// TwinCAT 3 PLC project PLC1
// Title: AutomationBaseClasses
// Company: PTW TU Darmstadt
// Author: Fabian Borst, Lukas Theisinger, Michael Frank, Tobias Lademann
// ProjectVersion: 1.1
// ProgramVersion: 3.1.4023.0
// libraries:
//   Tc2_ControllerToolbox, * (Beckhoff Automation GmbH)
//   Tc2_MBus, * (Beckhoff Automation GmbH)
//   Tc2_ModbusSrv, * (Beckhoff Automation GmbH)
//   Tc2_Standard, * (Beckhoff Automation GmbH)
//   Tc2_System, * (Beckhoff Automation GmbH)
//   Tc2_Utilities, * (Beckhoff Automation GmbH)
//   Tc3_Module, * (Beckhoff Automation GmbH)
// project tree:
//   DUTs/0 Base Data Structs/ E_SystemControlState.TcDUT, E_SystemOperatingState.TcDUT, ST_Control.TcDUT (not stored), ST_ControlState.TcDUT, ST_SensorState.TcDUT, ST_SetPointState.TcDUT, ST_SetSetPoint.TcDUT, ST_SystemState.TcDUT
//   DUTs/1 Actor Data Structs/DicreteValve/ E_DiscreteValveFeedbackMode.TcDUT, E_DiscreteValvePosition.TcDUT, ST_DiscreteValveDefaultParameters.TcDUT, ST_DiscreteValveState.TcDUT
//   DUTs/1 Actor Data Structs/MixingValve/ E_MixingValveControlMode.TcDUT, ST_MixingValveDefaultParameters.TcDUT, ST_MixingValveSetParameters.TcDUT
//   DUTs/1 Actor Data Structs/Pumps/ E_GrundfosMagna3ControlMode.TcDUT, ST_PumpGrundfosMagna3DefaultParameters.TcDUT, ST_PumpGrundfosMagna3Genibus.TcDUT, ST_PumpGrundfosMagna3SetParameters.TcDUT, ST_PumpGrundfosMagna3State.TcDUT
//   DUTs/2 Sensor Data Structs/ ST_ElectricityMeterState.TcDUT, ST_EmonioP3DefaultParameters.TcDUT, ST_EmonioP3State.TcDUT, ST_GasMeterDefaultParameters.TcDUT, ST_MollineC3HeatCounterState.TcDUT, ST_GasMeterState.TcDUT, ST_MollineC3HeatCounterDefaultParameters.TcDUT, ST_StarkMultical302HeatCounterState.TcDUT, ST_TemperatureSensorDefaultParameters.TcDUT (not stored)
//   DUTs/3 Utility Data Structs/ ST_RangeCheckDefaultParameters.TcDUT, ST_ClockDefaultParameters.TcDUT (not stored), ST_ClockState.TcDUT (not stored)
//   POUs/2 Sensors/ FB_ElectricityMeter_ABBA44113100.TcPOU, FB_ElectricityMeter_BergDCMI461WP.TcPOU, FB_ElectricityMeter_ABBA44213100.TcPOU, FB_EmonioP3.TcPOU, FB_GasMeter_Aerius_G4.TcPOU, FB_MollineEHeatCounter.TcPOU, FB_MollineUltramess403HeatCounter.TcPOU, FB_PressureSensor.TcPOU, FB_StarkMultical302HeatCounter.TcPOU, FB_TemperatureSensor_KL3214.TcPOU, FB_MollineC3HeatCounter.TcPOU, FB_TemperatureSensor.TcPOU
//   POUs/3 Utilities/0 Base/ FB_RangeCheck.TcPOU, FB_Clock.TcPOU, Limiter.TcPOU
//   POUs/3 Utilities/2 Profibus/ ConvertBitToByte.TcPOU, ConvertByteToBit.TcPOU (not stored), FB_Genibus.TcPOU, BufferIntToReal.TcPOU (not stored), BufferRealToReal.TcPOU (not stored), BufferUdintToReal.TcPOU
//   POUs/0 Base Classes/ FB_Actuator2Point.TcPOU, FB_ActuatorContinous.TcPOU, FB_Sensor.TcPOU, FB_SystemContinous.TcPOU
//   POUs/1 Actors/ FB_DiscreteValve.TcPOU, FB_PumpGrundfosMagna3.TcPOU, FB_MixingValve.TcPOU
//   POUs/3 Utilities/1 AI_AO/ FB_AnalogInput.TcPOU (not stored), FB_AnalogOutput.TcPOU
// real-time tasks:
//   TASK TaskMAIN: cycle T#10ms, priority 20, ADS port 350

// ---- DUTs/0 Base Data Structs/E_SystemControlState.TcDUT
{attribute 'qualified_only'}
{attribute 'strict'}
TYPE E_SystemControlState :
(
	automatic 	:= 0,
	algorithm	:= 1,
	manual		:= 2
);
END_TYPE

// ---- DUTs/0 Base Data Structs/E_SystemOperatingState.TcDUT
{attribute 'qualified_only'}
{attribute 'strict'}
TYPE E_SystemOperatingState :
(
	standby 	:= 0,
	rampUp		:= 1,
	rampDown	:= 2,
	operational	:= 3,
	working		:= 4
);
END_TYPE

// ---- DUTs/0 Base Data Structs/ST_ControlState.TcDUT
{attribute 'OPC.UA.DA.StructuredType' := '1'}
TYPE ST_ControlState :
STRUCT
	bStatusOn 		: BOOL; //status on / off
	sAccessMode		: STRING; //current access mode as string
	nAccessmode		: E_SystemControlState; //current access mode (1 = automatic, 2 = algorihm, 3 = manual)
END_STRUCT
END_TYPE

// ---- DUTs/0 Base Data Structs/ST_SensorState.TcDUT
{attribute 'OPC.UA.DA.StructuredType' := '1'}
TYPE ST_SensorState :
STRUCT
	fValue 		: REAL; //current value
	sUnit		: STRING; //current unit of sensor value
END_STRUCT
END_TYPE

// ---- DUTs/0 Base Data Structs/ST_SetPointState.TcDUT
{attribute 'OPC.UA.DA.StructuredType' := '1'}
TYPE ST_SetPointState :
STRUCT
	fOperatingPoint		: REAL; //current operating point
	fSetPoint			: REAL; //current set point
	sSetPointUnit		: STRING; //current set point unit
	sOperatingPointUnit : STRING; //current operating point unit 
	aSetPointLimits		: ARRAY[1..2] OF REAL; //lower and upper limit of setpoint
END_STRUCT
END_TYPE

// ---- DUTs/0 Base Data Structs/ST_SetSetPoint.TcDUT
{attribute 'OPC.UA.DA.StructuredType' := '1'}
TYPE ST_SetSetPoint :
STRUCT
	fSetPointAlgorithm		 : REAL; //set setpoint in percent 0.0 - 100.0
	fSetPointManual			 : REAL; //set setpoint in percent 0.0 - 100.0
END_STRUCT
END_TYPE

// ---- DUTs/0 Base Data Structs/ST_SystemState.TcDUT
{attribute 'OPC.UA.DA.StructuredType' := '1'}
TYPE ST_SystemState :
STRUCT
	sOperatingState : STRING; //operating state as string
	nOperatingState : E_SystemOperatingState; //operating state as integer
	bError : BOOL; //true if there is an error in any system component
END_STRUCT
END_TYPE

// ---- DUTs/1 Actor Data Structs/DicreteValve/E_DiscreteValveFeedbackMode.TcDUT
{attribute 'qualified_only'}
{attribute 'strict'}
TYPE E_DiscreteValveFeedbackMode :
(
	noFeedback := 0, //no feedback signal about valve position available
	openedFeedback := 1, //feedback signal if valve is open
	closedFeedback := 2, //feedback signal if valve is closed
	dualFeedback := 3 //feedback signal if valve is open/closed
);
END_TYPE

// ---- DUTs/1 Actor Data Structs/DicreteValve/E_DiscreteValvePosition.TcDUT
{attribute 'qualified_only'}
{attribute 'strict'}
TYPE E_DiscreteValvePosition :
(	
	noValidInformation := 0, //no information about position available
	moving := 1, //valve is moving
	closed := 2, //valve is closed
	open := 3 //valve is open
);
END_TYPE

// ---- DUTs/1 Actor Data Structs/DicreteValve/ST_DiscreteValveDefaultParameters.TcDUT
TYPE ST_DiscreteValveDefaultParameters :
STRUCT
	nFeedback : E_DiscreteValveFeedbackMode; //valve feedback mode as integer
END_STRUCT
END_TYPE

// ---- DUTs/1 Actor Data Structs/DicreteValve/ST_DiscreteValveState.TcDUT
TYPE ST_DiscreteValveState :
STRUCT
	nPosition : E_DiscreteValvePosition; //valve feedback mode as integer
END_STRUCT
END_TYPE

// ---- DUTs/1 Actor Data Structs/MixingValve/E_MixingValveControlMode.TcDUT
{attribute 'qualified_only'}
{attribute 'strict'}
TYPE E_MixingValveControlMode :
(
	position := 0, //control position
	heating := 1, //control temperature for heating application
	cooling := 2, //control temperature for cooling application
	thermalPower := 3 //control thermal power
);
END_TYPE

// ---- DUTs/1 Actor Data Structs/MixingValve/ST_MixingValveDefaultParameters.TcDUT
TYPE ST_MixingValveDefaultParameters:
STRUCT
	bFeedbackSignal : BOOL := TRUE; //true if valve gets a feedback signal for acual position
	fDefaultPosition : REAL := 0; //default position when bSetStatusOn = false
	fOffsetTerminal : REAL := 0; //voltage offset of terminal for input signal
	fControllerAmplification : LREAL := 0.265;
	tControllerIntegralTime : TIME := T#15S;
	fOutMaxLimit : LREAL := 100; //maximum output of controller
	fOutMinLimit : LREAL := 0; //minimum output of controller
	bARWOnIPartOnly : BOOL := TRUE; //if true, integration of I component stops, when integrator output reaches limit
	tTaskCycleTime	: TIME;
	tCtrlCycleTime	: TIME;
	aSetPointLimitsPosition	: ARRAY[1..2] OF REAL := [0,100]; //setpoint limits for position mode
	aSetPointLimitsTemperature : ARRAY[1..2] OF REAL := [0,100]; //setpoint limits for temperature mode
	aSetPointLimitsThermalPower : ARRAY[1..2] OF REAL := [-100,100]; //setpoint limits for heating and cooling power in kW
END_STRUCT
END_TYPE

// ---- DUTs/1 Actor Data Structs/MixingValve/ST_MixingValveSetParameters.TcDUT
{attribute 'OPC.UA.DA.StructuredType' := '1'}
TYPE ST_MixingValveSetParameters :
STRUCT
	nControlModeAlgorithm : E_MixingValveControlMode; //control mode in algorithm mode
	nControlModeManual : E_MixingValveControlMode; //control in manuel mode
END_STRUCT
END_TYPE

// ---- DUTs/1 Actor Data Structs/Pumps/E_GrundfosMagna3ControlMode.TcDUT
{attribute 'qualified_only'}
{attribute 'strict'}
TYPE E_GrundfosMagna3ControlMode :
(
	constantSpeed := 0, //constant speed control - 0.0 - 100.0 %
	constantTemperature_Heating := 1, //temperature control if flow is heated
	constantTemperature_Cooling := 2, //temperature control if flow is cooled
	temperatureDifference := 3, //temperature difference control
	pressureDifference := 4, //pressure difference control
	proportionalPressureControl := 5, //proportional pressure control
	thermalPower := 6 //thermal power control
);
END_TYPE

// ---- DUTs/1 Actor Data Structs/Pumps/ST_PumpGrundfosMagna3DefaultParameters.TcDUT
TYPE ST_PumpGrundfosMagna3DefaultParameters :
STRUCT
	bExternalTemperatureSensor 	: BOOL := TRUE; //pump measures beside the internal temperature als and external temperature
	bPumpBeforeApplication : BOOL := TRUE; //pump position before application
	fControllerAmplification : LREAL := 0.265;
	tControllerIntegralTime : TIME := T#15S;
	tTaskCycleTime	: TIME;
	tCtrlCycleTime	: TIME;	
	aSetPointLimits_constantSpeed : ARRAY[1..2] OF REAL := [0,100]; //degreeC
	aSetPointLimits_Temperature	: ARRAY[1..2] OF REAL := [0,100]; //degreeC
	aSetPointLimits_Pressure : ARRAY[1..2] OF REAL := [0,3]; //bar
	aSetPointLimitsThermalPower : ARRAY[1..2] OF REAL := [-100,100]; //setpoint limits for heating and cooling power in kW
	fMaximumVolumeFlowRate : REAL := 1.925; //default parameters for Magna3 25-40
	fNominalVolumeFlowRate : REAL := 0.000635; //default parameters for Magna3 25-40
	fMaximumPressureDifference : REAL := 40000; //default parameters for Magna3 25-40
END_STRUCT
END_TYPE

// ---- DUTs/1 Actor Data Structs/Pumps/ST_PumpGrundfosMagna3Genibus.TcDUT
TYPE ST_PumpGrundfosMagna3Genibus :
STRUCT
	SequenceNumber 	: BYTE;			(*SequenceNumber: Is the trigger, every time the value changes a new reply will be generated. *)
									(*For return telegram: values valid if Number matches request SquenceNumber*)
	DestAddress		: BYTE;			(*Address of GeniPro Slave, Broadcast = 16#FF*)
	Class			: BYTE;			(* no further Info provided*)
	OpLength		: BYTE; 		(* Operation and Length / for Reply Acknowledge and Length*)
	Data1			: BYTE;
	Data2			: BYTE;
	Data3			: BYTE;
	Data4			: BYTE;
	Data5			: BYTE;
END_STRUCT
END_TYPE

// ---- DUTs/1 Actor Data Structs/Pumps/ST_PumpGrundfosMagna3SetParameters.TcDUT
{attribute 'OPC.UA.DA.StructuredType' := '1'}
TYPE ST_PumpGrundfosMagna3SetParameters :
STRUCT
	nControlModeAlgorithm : E_GrundfosMagna3ControlMode; //control mode in algorithm mode
	nControlModeManual : E_GrundfosMagna3ControlMode; //control mode in manual mode
	bReset : BOOL; //resets errors and warnings
END_STRUCT
END_TYPE

// ---- DUTs/1 Actor Data Structs/Pumps/ST_PumpGrundfosMagna3State.TcDUT
{attribute 'OPC.UA.DA.StructuredType' := '1'}
TYPE ST_PumpGrundfosMagna3State :
STRUCT
	bRemoteControlOn : BOOL; //0 = control by pump, 1 = control by bus 	
	bError : BOOL; //true if pump shows an error
	bWarning : BOOL; //true if pump shows a warning
	sErrorMessage : STRING; //error code
	sWarningMessage : STRING; //warning code
	fVolumeFlowRate : REAL;
	sVolumeFlowRateUnit : STRING := 'm3/h';
	fTemperatureInternal : REAL; 
	sTemperatureInternalUnit : STRING := 'degreeC';
	fTemperatureExternal : REAL;
	sTemperatureExternalUnit : STRING := 'degreeC';
	fTemperatureDifference : REAL;
	sTemperatureDifferenceUnit: STRING := 'K';
	fPressureDifference : REAL;
	sPressureDifferenceUnit : STRING := 'Pa';
	fPowerElectric : REAL;
	sPowerElectricUnit : STRING := 'kW';
	fPowerHydraulic : REAL;
	sPowerHydraulicUnit : STRING := 'W';
	fPowerThermal : REAL;
	sPowerThermalUnit : STRING := 'W';
	fRotationalSpeed : REAL;
	sRotationalSpeedUnit : STRING := 'rpm';
END_STRUCT
END_TYPE

// ---- DUTs/2 Sensor Data Structs/ST_ElectricityMeterState.TcDUT
{attribute 'OPC.UA.DA.StructuredType' := '1'}
TYPE ST_ElectricityMeterState :
STRUCT
	fPower			: REAL;
	sPowerUnit		: STRING := 'kW';
	fWork			: REAL;
	sWorkUnit		: STRING := 'kWh';
END_STRUCT
END_TYPE

// ---- DUTs/2 Sensor Data Structs/ST_EmonioP3DefaultParameters.TcDUT
TYPE ST_EmonioP3DefaultParameters :
STRUCT
	fCalorificValue : REAL := 11.49;
END_STRUCT
END_TYPE

// ---- DUTs/2 Sensor Data Structs/ST_EmonioP3State.TcDUT
{attribute 'OPC.UA.DA.StructuredType' := '1'}
TYPE ST_EmonioP3State :
STRUCT
	fPower 					: REAL;
	sPowerUnit				: STRING := 'kW';
	fVoltage 				: REAL;
	sVoltageUnit			: STRING := 'V';
	fCurrent				: REAL;
	sCurrentUnit			: STRING := 'A';
	fEnergy					: REAL;
	sEnergyUnit				: STRING := 'kWh';
	fTemperature			: REAL;
	sTemperatureUnit		: STRING := 'degreeC';
	fPulse					: REAL;
	sPulse					: STRING := 'm^3';
	fPulseGasPower			: REAL;
	sPulseGasPower			: STRING := 'kW';
END_STRUCT
END_TYPE

// ---- DUTs/2 Sensor Data Structs/ST_GasMeterDefaultParameters.TcDUT
TYPE ST_GasMeterDefaultParameters :
STRUCT
	fCalorificValue : REAL := 11.49;
END_STRUCT
END_TYPE

// ---- DUTs/2 Sensor Data Structs/ST_MollineC3HeatCounterState.TcDUT
{attribute 'OPC.UA.DA.StructuredType' := '1'}
TYPE ST_MollineC3HeatCounterState :
STRUCT
	fVolume						: REAL;
	sVolumeUnit					: STRING := 'm3';
	fFeedTemperature			: REAL;
	sFeedTemperatureUnit		: STRING := 'degreeC';
	fReturnTemperature			: REAL;
	sReturnTemperatureUnit		: STRING := 'degreeC';
	fVolumeFlowRate				: REAL;
	sVolumeFlowRateUnit			: STRING := 'm3/h';
	fHeatEnergy					: REAL;
	sHeatEnergyUnit				: STRING := 'MWh';
	fHeatFlowRate				: REAL;
	sHeatFlowRateUnit			: STRING := 'kW';
	fTemperatureDifference		: REAL;
	sTemperatureDifferenceUnit 	: STRING := 'K';
END_STRUCT
END_TYPE

// ---- DUTs/2 Sensor Data Structs/ST_GasMeterState.TcDUT
{attribute 'OPC.UA.DA.StructuredType' := '1'}
TYPE ST_GasMeterState :
STRUCT
	fVolume					: REAL;
	sVolumeUnit				: STRING := 'm3';
	fTemperature			: REAL;
	sTemperatureUnit		: STRING := 'degreeC';
	fVolumeFlowRate			: REAL;
	sVolumeFlowRateUnit		: STRING := 'm3/h';
	fPower 					: REAL;
	sPowerUnit				: STRING := 'kW';
END_STRUCT
END_TYPE

// ---- DUTs/2 Sensor Data Structs/ST_MollineC3HeatCounterDefaultParameters.TcDUT
TYPE ST_MollineC3HeatCounterDefaultParameters:
STRUCT
	fSpecificHeatCapacity : REAL := 4.19;
END_STRUCT
END_TYPE

// ---- DUTs/2 Sensor Data Structs/ST_StarkMultical302HeatCounterState.TcDUT
{attribute 'OPC.UA.DA.StructuredType' := '1'}
TYPE ST_StarkMultical302HeatCounterState :
STRUCT
	fVolume						: REAL;
	sVolumeUnit					: STRING := 'm3';
	fFeedTemperature			: REAL;
	sFeedTemperatureUnit		: STRING := 'degreeC';
	fReturnTemperature			: REAL;
	sReturnTemperatureUnit		: STRING := 'degreeC';
	fVolumeFlowRate				: REAL;
	sVolumeFlowRateUnit			: STRING := 'm3/h';
	fHeatEnergy					: REAL;
	sHeatEnergyUnit				: STRING := 'MWh';
	fHeatFlowRate				: REAL;
	sHeatFlowRateUnit			: STRING := 'kW';
	fTemperatureDifference		: REAL;
	sTemperatureDifferenceUnit 	: STRING := 'K';
END_STRUCT
END_TYPE

// ---- DUTs/3 Utility Data Structs/ST_RangeCheckDefaultParameters.TcDUT
TYPE ST_RangeCheckDefaultParameters :
STRUCT
	fRestoreDifference : REAL; //difference to upper or lower limit to restore algorithm permission
	tTaskCycleTime : TIME;
	tCtrlCycleTime : TIME;
END_STRUCT
END_TYPE

// ---- POUs/2 Sensors/FB_ElectricityMeter_ABBA44113100.TcPOU
FUNCTION_BLOCK FB_ElectricityMeter_ABBA44113100
VAR_INPUT
	aElectricityMeterTelegramm	: ARRAY[1..cMBUS_MaxTelegrams] OF ST_MBus_Data2;
END_VAR
VAR_OUTPUT
	fWork : REAL; //Wh
	fPower : REAL; //W
END_VAR
VAR
	{attribute 'OPC.UA.DA' := '1'}
	sensorState : ST_ElectricityMeterState;
END_VAR

sensorState.fWork := STRING_TO_REAL(aElectricityMeterTelegramm[1].arrData[1].sValue)/1000;
sensorState.fPower := STRING_TO_REAL(aElectricityMeterTelegramm[2].arrData[1].sValue)/1000;

fWork := sensorState.fWork;
fPower := sensorState.fPower;

END_FUNCTION_BLOCK

// ---- POUs/2 Sensors/FB_ElectricityMeter_BergDCMI461WP.TcPOU
FUNCTION_BLOCK FB_ElectricityMeter_BergDCMI461WP
VAR_INPUT
	aElectricityMeterTelegramm	: ARRAY[1..cMBUS_MaxTelegrams] OF ST_MBus_Data2;
END_VAR
VAR_OUTPUT
	fWork : REAL; //Wh
	fPower : REAL; //W
END_VAR
VAR
	{attribute 'OPC.UA.DA' := '1'}
	sensorState : ST_ElectricityMeterState;
END_VAR

sensorState.fWork := STRING_TO_REAL(aElectricityMeterTelegramm[1].arrData[1].sValue)/1000;
sensorState.fPower := STRING_TO_REAL(aElectricityMeterTelegramm[1].arrData[2].sValue)/1000;

//set outputs
fWork := sensorState.fWork;
fPower := sensorState.fPower;

END_FUNCTION_BLOCK

// ---- POUs/2 Sensors/FB_ElectricityMeter_ABBA44213100.TcPOU
FUNCTION_BLOCK FB_ElectricityMeter_ABBA44213100
VAR_INPUT
	aElectricityMeterTelegramm	: ARRAY[1..cMBUS_MaxTelegrams] OF ST_MBus_Data2;
END_VAR
VAR_OUTPUT
	fWork : REAL; //Wh
	fPower : REAL; //W
END_VAR
VAR
	{attribute 'OPC.UA.DA' := '1'}
	sensorState : ST_ElectricityMeterState;
END_VAR

sensorState.fWork := STRING_TO_REAL(aElectricityMeterTelegramm[1].arrData[1].sValue)/1000;
sensorState.fPower := STRING_TO_REAL(aElectricityMeterTelegramm[2].arrData[2].sValue)/1000;

//set outputs
fWork := sensorState.fWork;
fPower := sensorState.fPower;

END_FUNCTION_BLOCK

// ---- POUs/2 Sensors/FB_EmonioP3.TcPOU
FUNCTION_BLOCK FB_EmonioP3
VAR_INPUT
	sIPAddr : STRING(15);
END_VAR
VAR_OUTPUT
	fPower : REAL; 			//kW
	fVoltage : REAL; 		//V
	fCurrent : REAL; 		//A
	fEnergy : REAL; 		//kWh
	fTemperature : REAL; 	//°C
	fPulse : REAL; 			//m^3
	fPulseGasPower : REAL;	//kW
	
	bErrorEM: BOOL;
	bErrorTemp: BOOL;
	bErrorPulse : BOOL;
END_VAR
VAR
	{attribute 'OPC.UA.DA' := '1'}
	sensorState : ST_EmonioP3State;
	
	localDefaultParameters : ST_EmonioP3DefaultParameters;
	
	fbEmonioElectricity : FB_MBReadRegs;
	fbEmonioTemperature : FB_MBReadRegs;
	fbEmonioPulse : FB_MBReadRegs;
	
	//timer to execute modbus fb
	Timer : TON;	
	bStartTimer : BOOL;
	bReadModbus : BOOL;
	
	arrInputRegsElectricity: ARRAY[0..13] OF WORD;			  // buffer for modbus fb electricity values
	arrInputRegsTemperature: ARRAY[0..1] OF WORD;			  // buffer for modbus fb temperature value
	arrInputRegsPulse: ARRAY[0..1] OF WORD;			  // buffer for modbus fb pulse value
	
    nErrIdEM: UDINT;
    nErrIdTemp: UDINT;
	nErrIdPulse: UDINT;
	
	//define arrays to convert from 16-bit word to real values
	PowerArray: ARRAY [0..1] OF WORD;
	VoltageArray: ARRAY [0..1] OF WORD;
	CurrentArray: ARRAY [0..1] OF WORD;
	EnergyArray: ARRAY [0..1] OF WORD;
	TemperatureArray: ARRAY [0..1] OF WORD;
	PulseArray: ARRAY [0..1] OF WORD;
	
	PowerInWatt : REAL; //helper variable to convert from W to kW
	
	//timer to execute modbus fb
	TimerGas : TON;	
	bStartTimerGas : BOOL;
	fPulseLastValue : REAL;
END_VAR

//Start and check timer for 2s interval
Timer(IN := bStartTimer,
	PT := T#2S);
bStartTimer := TRUE;
IF Timer.Q THEN
	bReadModbus := TRUE;
	bStartTimer := FALSE;	
END_IF

// Read Emonio via Modbus
fbEmonioElectricity(    
	sIPAddr := sIPAddr,   			//IP adress of the device
	nTCPPort := 502,				//Port number of the target device
	nUnitID := 255,					//Identification number of a serial sub-network device
	nQuantity  := 13,				//Number of input registers (data words) to be read
	nMBAddr := 300,					// Start address of the output registers to be read (word offset)
	cbLength := SIZEOF(arrInputRegsElectricity),
	pDestAddr := ADR(arrInputRegsElectricity),
	bExecute := bReadModbus,         // trigger
	tTimeout  := T#20S,
	bError => bErrorEM,				// Error handling
	nErrId => nErrIdEM				// Error handling 
);

fbEmonioTemperature(    
	sIPAddr := sIPAddr,   			//IP adress of the device
	nTCPPort := 502,				//Port number of the target device
	nUnitID := 255,					//Identification number of a serial sub-network device
	nQuantity  := 2,				//Number of input registers (data words) to be read
	nMBAddr := 500,					// Start address of the output registers to be read (word offset)
	cbLength := SIZEOF(arrInputRegsTemperature),
	pDestAddr := ADR(arrInputRegsTemperature),
	bExecute := bReadModbus,         // trigger
	tTimeout  := T#20S,
	bError => bErrorTemp,				// Error handling
	nErrId => nErrIdTemp				// Error handling 
);

fbEmonioPulse(    
	sIPAddr := sIPAddr,   			//IP adress of the device
	nTCPPort := 502,				//Port number of the target device
	nUnitID := 255,					//Identification number of a serial sub-network device
	nQuantity  := 2,				//Number of input registers (data words) to be read
	nMBAddr := 800,					// Start address of the output registers to be read (word offset)
	cbLength := SIZEOF(arrInputRegsPulse),
	pDestAddr := ADR(arrInputRegsPulse),
	bExecute := bReadModbus,         // trigger
	tTimeout  := T#20S,
	bError => bErrorPulse,				// Error handling
	nErrId => nErrIdPulse				// Error handling 
);

bReadModbus := FALSE;

//create arrays with word outputs
PowerArray[0] := arrInputRegsElectricity[4];
PowerArray[1] := arrInputRegsElectricity[5];
VoltageArray[0] := arrInputRegsElectricity[0];
VoltageArray[1] := arrInputRegsElectricity[1];
CurrentArray[0] := arrInputRegsElectricity[2];
CurrentArray[1] := arrInputRegsElectricity[3];
EnergyArray[0] := arrInputRegsElectricity[12];
EnergyArray[1] := arrInputRegsElectricity[13];
TemperatureArray[0] := arrInputRegsTemperature[0];
TemperatureArray[1] := arrInputRegsTemperature[1];
PulseArray[0] := arrInputRegsPulse[0];
PulseArray[1] := arrInputRegsPulse[1];

//convert word to real values
MEMCPY(ADR(PowerInWatt), ADR(PowerArray), 4);
sensorState.fPower := PowerInWatt/1000;
MEMCPY(ADR(sensorState.fVoltage), ADR(VoltageArray), 4);
MEMCPY(ADR(sensorState.fCurrent), ADR(CurrentArray), 4);
MEMCPY(ADR(sensorState.fEnergy), ADR(EnergyArray), 4);
MEMCPY(ADR(sensorState.fTemperature), ADR(TemperatureArray), 4);
MEMCPY(ADR(sensorState.fPulse), ADR(PulseArray), 4);

TimerGas(IN := bStartTimerGas,
	PT := T#30S);
bStartTimerGas := TRUE;

//overwrite last value durint init as long as last value remains zero
IF fPulseLastValue = 0 THEN
	fPulseLastValue := fPulse;
END_IF
IF TimerGas.Q THEN
	sensorState.fPulseGasPower := (fPulse-fPulseLastValue)*120*localDefaultParameters.fCalorificValue; //Gas power in kW
	fPulseLastValue := fPulse;
	bStartTimerGas := FALSE;	
END_IF

//define output variables
fPower := sensorState.fPower;
fVoltage := sensorState.fVoltage;
fCurrent := sensorState.fCurrent;
fEnergy := sensorState.fEnergy;
fTemperature := sensorState.fTemperature;
fPulse := sensorState.fPulse;
fPulseGasPower := sensorState.fPulseGasPower;

END_FUNCTION_BLOCK

// ---- POUs/2 Sensors/FB_GasMeter_Aerius_G4.TcPOU
FUNCTION_BLOCK FB_GasMeter_Aerius_G4
VAR_INPUT
	aGasmeterTelegramm	: ARRAY[1..cMBUS_MaxTelegrams] OF ST_MBus_Data2;
END_VAR
VAR_OUTPUT
	fVolumeFlowRate : REAL; //m3/h
	fTemperature : REAL; //°C
END_VAR
VAR
	{attribute 'OPC.UA.DA' := '1'}
	sensorState : ST_GasMeterState;
	
	localDefaultParameters : ST_GasMeterDefaultParameters;
END_VAR

sensorState.fTemperature := STRING_TO_REAL(aGasmeterTelegramm[1].arrData[3].sValue);
sensorState.fVolumeFlowRate := STRING_TO_REAL(aGasmeterTelegramm[1].arrData[2].sValue);
sensorState.fVolume := STRING_TO_REAL(aGasmeterTelegramm[1].arrData[1].sValue);
sensorState.fPower := sensorState.fVolumeFlowRate*localDefaultParameters.fCalorificValue; //calculate Power in kW

//set outputs
fVolumeFlowRate := sensorState.fVolume;
fTemperature := sensorState.fTemperature;

END_FUNCTION_BLOCK

// ---- POUs/2 Sensors/FB_MollineEHeatCounter.TcPOU
FUNCTION_BLOCK FB_MollineEHeatCounter
VAR_INPUT
	aHeatCounterTelegramm : ARRAY[1..cMBUS_MaxTelegrams] OF ST_MBus_Data2;
END_VAR
VAR_OUTPUT
	fFeedTemperature : REAL; //°C
	fReturnTemperature : REAL; //°C
	fVolumeFlowRate : REAL; //m3/h
	fHeatFlowRate : REAL; //kW
END_VAR
VAR
	{attribute 'OPC.UA.DA' := '1'}
	sensorState : ST_MollineC3HeatCounterState;
END_VAR

//set sensor state
sensorState.fVolume := STRING_TO_REAL(aHeatCounterTelegramm[1].arrData[3].sValue);
sensorState.fFeedTemperature := STRING_TO_REAL(aHeatCounterTelegramm[1].arrData[7].sValue);
sensorState.fReturnTemperature := STRING_TO_REAL(aHeatCounterTelegramm[1].arrData[8].sValue);
sensorState.fVolumeFlowRate := STRING_TO_REAL(aHeatCounterTelegramm[1].arrData[6].sValue);
sensorState.fHeatEnergy := STRING_TO_REAL(aHeatCounterTelegramm[1].arrData[2].sValue)/1000000;
sensorState.fTemperatureDifference := STRING_TO_REAL(aHeatCounterTelegramm[1].arrData[9].sValue);

//calculate fHeatFlowRate because heat meter does not measure negative flows
sensorState.fHeatFlowRate := sensorState.fVolumeFlowRate/3.6*4.19*sensorState.fTemperatureDifference;

//set outputs
fFeedTemperature := sensorState.fFeedTemperature;
fReturnTemperature := sensorState.fReturnTemperature;
fVolumeFlowRate := sensorState.fVolumeFlowRate;
fHeatFlowRate := sensorState.fHeatFlowRate;

END_FUNCTION_BLOCK

// ---- POUs/2 Sensors/FB_MollineUltramess403HeatCounter.TcPOU
FUNCTION_BLOCK FB_MollineUltramess403HeatCounter
VAR_INPUT
	aHeatCounterTelegramm : ARRAY[1..cMBUS_MaxTelegrams] OF ST_MBus_Data2;
END_VAR
VAR_OUTPUT
	fFeedTemperature : REAL; //°C
	fReturnTemperature : REAL; //°C
	fVolumeFlowRate : REAL; //m3/h
	fHeatFlowRate : REAL; //kW
END_VAR
VAR
	{attribute 'OPC.UA.DA' := '1'}
	sensorState : ST_MollineC3HeatCounterState;
END_VAR

//set sensor state
sensorState.fVolume := STRING_TO_REAL(aHeatCounterTelegramm[1].arrData[5].sValue);
sensorState.fFeedTemperature := STRING_TO_REAL(aHeatCounterTelegramm[1].arrData[11].sValue);
sensorState.fReturnTemperature := STRING_TO_REAL(aHeatCounterTelegramm[1].arrData[12].sValue);
sensorState.fVolumeFlowRate := STRING_TO_REAL(aHeatCounterTelegramm[1].arrData[17].sValue);
sensorState.fHeatEnergy := STRING_TO_REAL(aHeatCounterTelegramm[1].arrData[2].sValue)/1000000;
sensorState.fTemperatureDifference := STRING_TO_REAL(aHeatCounterTelegramm[1].arrData[13].sValue);

//calculate fHeatFlowRate because heat meter does not measure negative flows
sensorState.fHeatFlowRate := sensorState.fVolumeFlowRate/3.6*4.19*sensorState.fTemperatureDifference;

//set outputs
fFeedTemperature := sensorState.fFeedTemperature;
fReturnTemperature := sensorState.fReturnTemperature;
fVolumeFlowRate := sensorState.fVolumeFlowRate;
fHeatFlowRate := sensorState.fHeatFlowRate;

END_FUNCTION_BLOCK

// ---- POUs/2 Sensors/FB_PressureSensor.TcPOU
FUNCTION_BLOCK FB_PressureSensor EXTENDS FB_Sensor
VAR_INPUT
END_VAR
VAR_OUTPUT
	fPressure : REAL; //measured pressure in bar
END_VAR
VAR	
	//I/O-Links
	nPressure_IN AT %I* : INT;
END_VAR

METHOD GetState_AI : BOOL
VAR_INPUT
END_VAR
VAR
END_VAR
// scaling to [0,6000]
fPressure := (INT_TO_REAL(nPressure_IN))*0.1831/1000 ;

//sensor state
sensorState.fValue := fPressure;
sensorState.sUnit := 'bar';
END_METHOD

END_FUNCTION_BLOCK

// ---- POUs/0 Base Classes/FB_Sensor.TcPOU
FUNCTION_BLOCK ABSTRACT FB_Sensor
VAR_INPUT
END_VAR
VAR_OUTPUT
END_VAR
VAR
	{attribute 'OPC.UA.DA' := '1'}
	sensorState : ST_SensorState;
END_VAR

END_FUNCTION_BLOCK

// ---- POUs/2 Sensors/FB_StarkMultical302HeatCounter.TcPOU
FUNCTION_BLOCK FB_StarkMultical302HeatCounter
VAR_INPUT
	aHeatCounterTelegramm : ARRAY[1..cMBUS_MaxTelegrams] OF ST_MBus_Data2;
END_VAR
VAR_OUTPUT
	fFeedTemperature : REAL; //°C
	fReturnTemperazure : REAL; //°C
	fVolumeFlowRate : REAL; //m3/h
END_VAR
VAR
	{attribute 'OPC.UA.DA' := '1'}
	sensorState : ST_StarkMultical302HeatCounterState;
END_VAR

//set sensor state
sensorState.fVolume := STRING_TO_REAL(aHeatCounterTelegramm[1].arrData[6].sValue);
sensorState.fFeedTemperature := STRING_TO_REAL(aHeatCounterTelegramm[1].arrData[9].sValue);
sensorState.fReturnTemperature := STRING_TO_REAL(aHeatCounterTelegramm[1].arrData[10].sValue);
sensorState.fVolumeFlowRate := STRING_TO_REAL(aHeatCounterTelegramm[1].arrData[14].sValue);
sensorState.fHeatEnergy := STRING_TO_REAL(aHeatCounterTelegramm[1].arrData[2].sValue)/1000000;
sensorState.fTemperatureDifference := STRING_TO_REAL(aHeatCounterTelegramm[1].arrData[11].sValue);

//calculate fHeatFlowRate because heat meter does not measure negative flows
sensorState.fHeatFlowRate := sensorState.fVolumeFlowRate/3.6*4.19*sensorState.fTemperatureDifference;

//set outputs
fFeedTemperature := sensorState.fFeedTemperature;
fReturnTemperazure := sensorState.fReturnTemperature;
fVolumeFlowRate := sensorState.fVolumeFlowRate;

END_FUNCTION_BLOCK

// ---- POUs/2 Sensors/FB_TemperatureSensor_KL3214.TcPOU
FUNCTION_BLOCK FB_TemperatureSensor_KL3214 EXTENDS FB_Sensor
VAR_INPUT
END_VAR
VAR_OUTPUT
	fTemperature : REAL; //measured temperature in degreeC
END_VAR
VAR	
	//I/O-Links
	temperature_IN AT %I* : INT;
END_VAR

METHOD GetState_AI : BOOL
VAR_INPUT
END_VAR
VAR
END_VAR
// conversion with 0.1 resolution
fTemperature := (INT_TO_REAL(temperature_IN))*0.1;

//sensor state
sensorState.fValue := fTemperature;
sensorState.sUnit := 'degreeC';
END_METHOD

END_FUNCTION_BLOCK

// ---- POUs/3 Utilities/0 Base/FB_RangeCheck.TcPOU
FUNCTION_BLOCK FB_RangeCheck
VAR_INPUT
	fInput : REAL;
	fLowerLimit : REAL; //lower limit of permission range
	fUpperLimit : REAL; //upper limit of permission range
END_VAR
VAR_OUTPUT
	bPermission : BOOL := TRUE;
END_VAR
VAR
	localDefaultParameters : ST_RangeCheckDefaultParameters;	

	Controller_UpperLimit : FB_CTRL_2POINT;
	Controller_LowerLimit : FB_CTRL_2POINT;
	Controller_Parameters : ST_CTRL_2POINT_PARAMS;	
END_VAR

Controller_Parameters.fHysteresisRange := localDefaultParameters.fRestoreDifference;
Controller_Parameters.tCtrlCycleTime := localDefaultParameters.tCtrlCycleTime;
Controller_Parameters.tTaskCycleTime := localDefaultParameters.tTaskCycleTime;

Controller_UpperLimit(fSetpointValue := fUpperLimit - localDefaultParameters.fRestoreDifference/2,
	fActualValue := fInput,
	eMode := eCTRL_MODE_ACTIVE,
	stParams := Controller_Parameters);
	
Controller_LowerLimit(fSetpointValue := fInput,
	fActualValue := fLowerLimit + localDefaultParameters.fRestoreDifference/2,
	eMode := eCTRL_MODE_ACTIVE,
	stParams := Controller_Parameters);
	
bPermission := Controller_UpperLimit.bOut AND Controller_LowerLimit.bOut;

PROPERTY ST_DefaultParameters : REFERENCE TO ST_RangeCheckDefaultParameters
SET
localDefaultParameters := ST_DefaultParameters;
END_SET
END_PROPERTY

END_FUNCTION_BLOCK

// ---- POUs/3 Utilities/0 Base/FB_Clock.TcPOU
FUNCTION_BLOCK FB_Clock
VAR_INPUT
END_VAR
VAR_OUTPUT
	stClockState : ST_ClockState;
END_VAR
VAR
	localDefaultParameters : ST_ClockDefaultParameters;

	Clock				: FB_CTRL_GET_SYSTEM_TIME;
	Clock_Parameters	: ST_CTRL_GET_SYSTEM_TIME_PARAMS;
END_VAR

Clock_Parameters.tTaskCycleTime	:= localDefaultParameters.tTaskCycleTime;
Clock_Parameters.tCtrlCycleTime	:= localDefaultParameters.tCtrlCycleTime;

Clock(stParams := Clock_Parameters);

stClockState.sintMonth		:= WORD_TO_SINT(Clock.stSystemTime.wMonth);
stClockState.sintDay		:= WORD_TO_SINT(Clock.stSystemTime.wDay);
stClockState.sintWeekday	:= WORD_TO_SINT(Clock.stSystemTime.wDayOfWeek);
stClockState.fHour			:= WORD_TO_REAL(Clock.stSystemTime.wHour) + WORD_TO_REAL(Clock.stSystemTime.wMinute) / 60;

PROPERTY ST_DefaultParameters : REFERENCE TO ST_ClockDefaultParameters
SET
localDefaultParameters := ST_DefaultParameters;
END_SET
END_PROPERTY

END_FUNCTION_BLOCK

// ---- POUs/3 Utilities/2 Profibus/ConvertBitToByte.TcPOU
FUNCTION ConvertBitToByte : BYTE
VAR_INPUT
	dataBit : ARRAY[0..7] OF BOOL;
END_VAR
VAR
	dataByte : BYTE;
END_VAR

dataByte.0 := dataBit[0];
dataByte.1 := dataBit[1];
dataByte.2 := dataBit[2];
dataByte.3 := dataBit[3];
dataByte.4 := dataBit[4];
dataByte.5 := dataBit[5];
dataByte.6 := dataBit[6];
dataByte.7 := dataBit[7];

ConvertBitToByte := dataByte;

END_FUNCTION

// ---- POUs/3 Utilities/2 Profibus/FB_Genibus.TcPOU
FUNCTION_BLOCK FB_Genibus
VAR_INPUT
	Reply						:  POINTER TO ST_PumpGrundfosMagna3Genibus; 	//This is mapped to PB_DPV0 Module 43 "DirectDataReply"
	Request 					:  POINTER TO ST_PumpGrundfosMagna3Genibus; 	//This is mapped to PB_DPV0 Module 42 "DirectDataRequest"
END_VAR
VAR_OUTPUT
	preciseInternalTemperature 	:	REAL; //Here the resulting precise Value will be stored
END_VAR
VAR
	bInitialize					: BOOL := FALSE;
	last_request				: TIME;
END_VAR

(* Initialize PROGRAM*)
IF bInitialize = FALSE THEN
	Request^.DestAddress 		:= 16#FF; 		(* Set destination to "Broadcast"*)
	Request^.Class				:= 16#0B;		(* Select Class 11 as Provided by Grundfos*)
	Request^.OpLength			:= 16#01;		(*Operation = GET (0), Length = 1*)
	Request^.Data1				:= 16#22;		(* ID = 34 (Probably for internal Temperature) ||  Volumenstrom ID = 53 (in hex: 16#35) *)
	Request^.SequenceNumber 	:= 1;			(*Trigger first Request*)

	bInitialize := TRUE;

	last_request := TIME();

ELSE

(*Programm is now ready for reading*)
	IF Reply^.SequenceNumber = Request^.SequenceNumber THEN (*Sequence Number of Incoming data has to match that of request!*)

		IF Reply^.OpLength = 16#02 THEN (* otherwise an error occured ! *)
			preciseInternalTemperature := (Reply^.Data1*255+Reply^.Data2)*0.01-273.16;  (*Data1 contains the Highbyte, Data2 the Lowbyte. Resulting Value is in [K], substract 273.16 for getting [°C]*)
		END_IF

		IF  TIME()-last_request >= T#1s THEN
			Request^.SequenceNumber := Request^.SequenceNumber +1;	(* Increase SequenceNumber to trigger next Request*)
			last_request := TIME();
		END_IF

	END_IF
END_IF

END_FUNCTION_BLOCK

// ---- POUs/0 Base Classes/FB_Actuator2Point.TcPOU
FUNCTION_BLOCK ABSTRACT FB_Actuator2Point
VAR_INPUT
	bSetStatusOnAutomatic : BOOL; //turn actor on
	bAlgorithmPermission : BOOL; //is true if control by algorithm is allowed
END_VAR
VAR_OUTPUT
	bStatusOn : BOOL; //true if actor is on
END_VAR
VAR
	{attribute 'OPC.UA.DA' := '1'}
	control : ST_Control;
	{attribute 'OPC.UA.DA' := '1'}
	controlState : ST_ControlState;

	//internal variables
	bSetStatusOn : BOOL; //actual internal value to switch on 
END_VAR

METHOD PROTECTED SelectControlMode : BOOL
VAR_INPUT
END_VAR
VAR
END_VAR
//change access mode
IF control.bManualModeActivated THEN
	controlState.nAccessmode := E_SystemControlState.manual;
	controlState.sAccessMode := 'manual';
	bSetStatusOn := control.bSetStatusOnManual;
ELSIF control.bAlgorithmModeActivated AND bAlgorithmPermission THEN
	controlState.nAccessmode := E_SystemControlState.algorithm;
	controlState.sAccessMode := 'algorithm';
	bSetStatusOn := control.bSetStatusOnAlgorithm;
ELSE
	controlState.nAccessmode := E_SystemControlState.automatic;
	controlState.sAccessMode := 'automatic';
	bSetStatusOn := bSetStatusOnAutomatic;
END_IF
END_METHOD

END_FUNCTION_BLOCK

// ---- POUs/0 Base Classes/FB_ActuatorContinous.TcPOU
FUNCTION_BLOCK ABSTRACT FB_ActuatorContinous EXTENDS FB_Actuator2Point
VAR_INPUT
	fSetPointAutomatic	: REAL; //setpoint in automatic mode
END_VAR
VAR_OUTPUT
	fOperatingPoint : REAL; //operating point
END_VAR
VAR
	{attribute 'OPC.UA.DA' := '1'}
	setSetPoint : ST_SetSetPoint;
	{attribute 'OPC.UA.DA' := '1'}
	setPointState : ST_SetPointState;
	
	//internal variables
	fSetPoint	    : REAL; //actual set setpoint
	aSetPointLimits	: ARRAY[1..2] OF REAL; //control mode depending setpoint limits that are set by abstract method SetSetPointLimits() in child class 
END_VAR

METHOD MAIN : BOOL
VAR_INPUT
END_VAR
SelectControlMode();
SelectSetPoint();
SetSetPointLimits();
SetPointCheck();
END_METHOD

METHOD PROTECTED SelectSetPoint : BOOL
VAR_INPUT
END_VAR
IF control.bManualModeActivated THEN
	fsetPoint := setSetPoint.fSetPointManual;
ELSIF control.bAlgorithmModeActivated AND bAlgorithmPermission THEN
	fsetPoint := setSetPoint.fSetPointAlgorithm;
ELSE
	fsetPoint := fSetPointAutomatic;
END_IF
END_METHOD

METHOD PRIVATE SetPointCheck : BOOL
VAR
END_VAR
fSetPoint := MAX(fSetPoint, aSetPointLimits[1]);
fSetPoint := MIN(fSetPoint, aSetPointLimits[2]);
END_METHOD

METHOD PROTECTED ABSTRACT SetSetPointLimits : BOOL
VAR_INPUT
END_VAR
//set control mode depending setpoint limits -> aSetPointLimits
END_METHOD

END_FUNCTION_BLOCK

// ---- POUs/0 Base Classes/FB_SystemContinous.TcPOU
FUNCTION_BLOCK ABSTRACT FB_SystemContinous EXTENDS FB_ActuatorContinous
VAR_INPUT
END_VAR
VAR_OUTPUT
END_VAR
VAR
	{attribute 'OPC.UA.DA' := '1'}
	systemState : ST_SystemState;
END_VAR

METHOD PROTECTED ABSTRACT CheckError : BOOL
VAR_INPUT
END_VAR
VAR_OUTPUT
	bError : BOOL;
END_VAR
END_METHOD

METHOD MAIN : BOOL // Method that calls all needed function block methods
VAR_INPUT
END_VAR
SUPER^.MAIN();
SetState();
SystemFlowControl();
END_METHOD

METHOD PROTECTED ABSTRACT Operational : BOOL
VAR_INPUT
END_VAR
VAR_OUTPUT
	bSwitchToWorking : BOOL := FALSE;
END_VAR
END_METHOD

METHOD PROTECTED ABSTRACT RampDown : BOOL
VAR_INPUT
END_VAR
VAR_OUTPUT
	bRampDownFinished : BOOL := FALSE;
END_VAR
END_METHOD

METHOD PROTECTED ABSTRACT RampUp : BOOL
VAR_INPUT
END_VAR
VAR_OUTPUT
	bRampUpFinished : BOOL := FALSE;
END_VAR
END_METHOD

METHOD PROTECTED ABSTRACT  SetSetPointLimits : BOOL
VAR_INPUT
END_VAR
END_METHOD

METHOD PROTECTED ABSTRACT SetState : BOOL
VAR_INPUT
END_VAR
VAR_OUTPUT
END_VAR
END_METHOD

METHOD SystemFlowControl : INT
VAR_INPUT
END_VAR
VAR_INST
	nState : E_SystemOperatingState := E_SystemOperatingState.standby; //actual state number
	bSwitchState : BOOL := FALSE;
	bSystemError : BOOL := FALSE;
END_VAR
CheckError(bError => bSystemError);
systemState.bError := bSystemError;

IF NOT bSystemError THEN
	CASE nState OF
		E_SystemOperatingState.standby:
			systemState.sOperatingState := 'standby';
			bSwitchState := FALSE;
			//if turned on switch to ramp-up
			IF(bSetStatusOn) THEN
				nState := E_SystemOperatingState.rampUp;
			END_IF
		E_SystemOperatingState.rampUp:
			systemState.sOperatingState := 'ramp-up';
			RampUp(bRampUpFinished => bSwitchState);
			//if turned off switch to ramp-down
			IF(NOT bSetStatusOn) THEN
				nState := E_SystemOperatingState.rampDown;
			//if ramp-up finished switch to operational
			ELSIF(bSwitchState) THEN
				nState := E_SystemOperatingState.operational;
			END_IF
		E_SystemOperatingState.operational:
			systemState.sOperatingState := 'operational';
			Operational(bSwitchToWorking => bSwitchState);
			//if turned off switch to ramp-down
			IF(NOT bSetStatusOn) THEN
				nState := E_SystemOperatingState.rampDown;
			//switch to working if desired
			ELSIF(bSwitchState) THEN
				nState := E_SystemOperatingState.working;
			END_IF
		E_SystemOperatingState.working:
			systemState.sOperatingState := 'working';
			Working(bSwitchToOperational => bSwitchState);
			//if turned off switch to ramp-down
			IF(NOT bSetStatusOn) THEN
				nState := E_SystemOperatingState.rampDown;
			//switch to operational if desired
			ELSIF(bSwitchState) THEN
				nState := E_SystemOperatingState.operational;
			END_IF
		E_SystemOperatingState.rampDown:
			systemState.sOperatingState := 'ramp-down';
			RampDown(bRampDownFinished => bSwitchState);
			//if turned on switch to ramp-up
			IF(bSetStatusOn) THEN
				nState := E_SystemOperatingState.rampUp;
			//if ramp-down finished switch to standby
			ELSIF(bSwitchState) THEN
				nState := E_SystemOperatingState.standby;
			END_IF
	END_CASE
ELSE
	RampDown(bRampDownFinished => bSwitchState);
	IF bSwitchState THEN
		systemState.sOperatingState := 'standby';
		nState := E_SystemOperatingState.standby;
	ELSE
		systemState.sOperatingState := 'ramp-down';	
		nState := E_SystemOperatingState.rampDown;		
	END_IF
	
END_IF
systemState.nOperatingState := nState;
END_METHOD

METHOD PROTECTED ABSTRACT Working : BOOL
VAR_INPUT
END_VAR
VAR_OUTPUT
	bSwitchToOperational : BOOL := FALSE;
END_VAR
END_METHOD

END_FUNCTION_BLOCK

// ---- POUs/1 Actors/FB_DiscreteValve.TcPOU
FUNCTION_BLOCK FB_DiscreteValve EXTENDS FB_Actuator2Point
VAR_INPUT
END_VAR
VAR_OUTPUT
	{attribute 'OPC.UA.DA' := '1'}
	localState : ST_DiscreteValveState;
END_VAR
VAR
	//default parameters
	localDefaultParameters : ST_DiscreteValveDefaultParameters;	

	//I/O Links
	bSetStatusOn_OUT 	AT %Q* : BOOL := FALSE;
	bStatusOn_IN		AT %I* : BOOL := FALSE; //True if valve is 100 % open
	bStatusOff_IN		AT %I* : BOOL := FALSE; //True if valve is 100 % closed
	(* NOTE: 
	If valve provides only one feedback signal, bStatusOn_IN must be linked to the terminal. 
	If valve provides feedback signals for reaching open/closed position, bStatusOff_IN must be also linked to the terminal.
	If there is no feedback signal, no input signal must be linked.
	The correct mode must be declared using localDefaultParameters.nFeedback
	*)
END_VAR

SelectControlMode();

METHOD GetState_BI : BOOL
VAR_INPUT
END_VAR
CASE localDefaultParameters.nFeedback OF
	1: //feedback - valve opened
	controlState.bStatusOn := bStatusOn_IN;
	IF bStatusOn_IN THEN
		localState.nPosition := 3;
	ELSE
		localState.nPosition := 0;
	END_IF 
	
	2: //feedback - valve closed
	controlState.bStatusOn := NOT bStatusOff_IN;
	IF bStatusOff_IN THEN
		localState.nPosition := 2;
	ELSE
		localState.nPosition := 0;
	END_IF 

	3: //feedback - both states
	controlState.bStatusOn := bStatusOn_IN;
	IF bStatusOff_IN THEN
		localState.nPosition := 2;
	ELSIF bStatusOn_IN THEN
		localState.nPosition := 3;
	ELSE
		localState.nPosition := 1;
	END_IF
ELSE
	localState.nPosition := 0; //no valid information
	controlState.bStatusOn := 0; //no valid information
END_CASE
bStatusOn := controlState.bStatusOn;
END_METHOD

METHOD SetState_BO : BOOL
VAR_INPUT
END_VAR
VAR
END_VAR
bSetStatusOn_OUT := bSetStatusOn;
END_METHOD

METHOD SetState_Inverted_BO : BOOL
VAR_INPUT
END_VAR
bSetStatusOn_OUT := NOT bSetStatusOn;
END_METHOD

PROPERTY ST_DefaultParameters : REFERENCE TO ST_DiscreteValveDefaultParameters
SET
localDefaultParameters := ST_DefaultParameters;
END_SET
END_PROPERTY

END_FUNCTION_BLOCK

// ---- POUs/1 Actors/FB_PumpGrundfosMagna3.TcPOU
FUNCTION_BLOCK FB_PumpGrundfosMagna3 EXTENDS FB_ActuatorContinous
VAR_INPUT
	nControlModeAutomatic : E_GrundfosMagna3ControlMode;
	fExternalValue : REAL; //external value for control, e. g. temperature, temperature difference volume flow rate
	fThermalPowerExternal : REAL; //external heat power in kW
END_VAR
VAR_OUTPUT
	bError : BOOL; //true if pump is in error
	fTemperatureInternal : REAL; //internal temperature (e.g. for temperature controlling valves)
	fTemperatureExternal : REAL; //external temperature (e.g. for temperature controlling valves)
	fVolumeFlowRate : REAL;
END_VAR
VAR
	{attribute 'OPC.UA.DA' := '1'}
	localSetParameters : ST_PumpGrundfosMagna3SetParameters;
	{attribute 'OPC.UA.DA' := '1'}
	localState : ST_PumpGrundfosMagna3State;
	
	//default parameters
	localDefaultParameters : ST_PumpGrundfosMagna3DefaultParameters;
	
	//I/O links
	StatusModule_IN						AT %I* : ARRAY [0..5] OF BYTE;
	nAlarmCode_IN						AT %I* : USINT;
	nWarningCode_IN						AT %I* : USINT;
	fVolumeFlowRate_IN 					AT %I* : UDINT; //m^3/h volume flow rate from pump
	fPressureDifference_IN	 			AT %I* : UDINT; //pa = 10^-5 bar
	fPowerElectric_IN					AT %I* : UDINT; //kW
	fActualSetpoint_IN					AT %I* : UDINT; //%
	fRotationalSpeed_IN	 				AT %I* : UDINT; //rpm
	fTemperatureExternal_IN 			AT %I* : UDINT; //°C external temperature from sensor connected to pump
	fTemperatureDifference_IN			AT %I* : UDINT; //°C
	fPowerThermal_IN	 				AT %I* : UDINT; //W
	ControlModule_OUT 					AT %Q* : ARRAY [0..4] OF BYTE;
	
	//Genibus
	Genibus : FB_Genibus;
	stTemperatureInternal_Genibus_Reply 	AT %I* : ST_PumpGrundfosMagna3Genibus;
	stTemperatureInternal_Genibus_Request	AT %Q* : ST_PumpGrundfosMagna3Genibus;
	
	//controllers
	PI_Controller				: FB_CTRL_PI; 
	PI_Controller_Parameters 	: ST_CTRL_PI_PARAMS;
	fSetpointValue 				: LREAL; //internal setpoint value (is switched depending on heating/cooling application)
	fActualValue 				: LREAL; //internal setpoint value (is switched depending on heating/cooling application)
	fAct 						: REAL; //actual measured value from internal pump sensor or external sensor
		
	//internal variables:
	nControlMode 			: E_GrundfosMagna3ControlMode; //actual pump control mode
	fSetPoint_controlled 	: REAL; //controlled setpoint
	statusModule0Bits 		: ARRAY[0..7] OF BOOL;
	tmp 					: STRING;
	controlModule0Bits 		: ARRAY[0..7] OF BOOL;
END_VAR

MAIN();
SelectLocalControlMode();
CalculateHydraulicPower();
LocalControl();
Genibus(Reply := ADR(stTemperatureInternal_Genibus_Reply), Request := ADR(stTemperatureInternal_Genibus_Request));

METHOD PRIVATE CalculateHydraulicPower : REAL
VAR_INPUT
END_VAR
localState.fPowerHydraulic := localState.fPressureDifference*localState.fVolumeFlowRate;
END_METHOD

METHOD GetState_Profibus : BOOL
VAR_INPUT
END_VAR
VAR
END_VAR
statusModule0Bits := ConvertByteToBit(dataByte:=StatusModule_IN[0]);

//control state
controlState.bStatusOn := statusModule0Bits[1];
bStatusOn := controlState.bStatusOn;

//setpoint state
setPointState.fOperatingPoint := BufferUdintToReal(raw_input := fActualSetpoint_IN);
fOperatingPoint := setPointState.fOperatingPoint;
setPointState.sOperatingPointUnit := 'percent';

//local state
localState.bError := statusModule0Bits[2];
localState.bWarning := statusModule0Bits[3];
bError := localState.bError;
localState.sErrorMessage := CONCAT('Alarm code: ',INT_TO_STRING(nAlarmCode_IN));
localState.sWarningMessage := CONCAT('Warning code: ',INT_TO_STRING(nWarningCode_IN));
localState.bRemoteControlOn := statusModule0Bits[0];
localState.fVolumeFlowRate := BufferUdintToReal(raw_input := fVolumeFlowRate_IN);
localState.fTemperatureInternal := BufferRealToReal(raw_input := Genibus.preciseInternalTemperature);
fTemperatureInternal := localState.fTemperatureInternal;
IF localDefaultParameters.bExternalTemperatureSensor THEN //Set external temperature and temperature difference if temperature sensor is connected
	localState.fTemperatureExternal := BufferUdintToReal(raw_input := fTemperatureExternal_IN);
	fTemperatureExternal := localState.fTemperatureExternal;
	localState.fTemperatureDifference := localState.fTemperatureInternal-localState.fTemperatureExternal;
END_IF;
localState.fPressureDifference := BufferUdintToReal(raw_input := fPressureDifference_IN);
localState.fPowerElectric := BufferUdintToReal(raw_input := fPowerElectric_IN)/1000; //W->kW
localState.fPowerThermal := BufferUdintToReal(raw_input := fPowerThermal_IN);
localState.fRotationalSpeed := BufferUdintToReal(raw_input := fRotationalSpeed_IN);
fVolumeFlowRate := localState.fVolumeFlowRate;
END_METHOD

METHOD PRIVATE LocalControl : BOOL
VAR_INPUT
END_VAR
VAR
END_VAR
//set control parameters
PI_Controller_Parameters.fKp 				:= localDefaultParameters.fControllerAmplification;
PI_Controller_Parameters.tTn 				:= localDefaultParameters.tControllerIntegralTime;
PI_Controller_Parameters.fOutMaxLimit		:= 100.0;
PI_Controller_Parameters.fOutMinLimit		:= 0.0;
PI_Controller_Parameters.tTaskCycleTime		:= localDefaultParameters.tTaskCycleTime;
PI_Controller_Parameters.tCtrlCycleTime		:= localDefaultParameters.tCtrlCycleTime;
PI_Controller_Parameters.bARWOnIPartOnly	:= TRUE;

//check which actual value should be used depending on control mode, external temperature sensor and pump place
CASE nControlMode OF
	1,2: //constant temperature control
	IF localDefaultParameters.bPumpBeforeApplication THEN
		IF localDefaultParameters.bExternalTemperatureSensor THEN
			fAct := localState.fTemperatureExternal;
		ELSE
			fAct := fExternalValue;
		END_IF
	ELSE
		fAct := localState.fTemperatureInternal;		
	END_IF
	
	3: //temperature difference control
	fAct := localState.fTemperatureDifference;
	IF localDefaultParameters.bPumpBeforeApplication AND NOT localDefaultParameters.bExternalTemperatureSensor THEN
		fAct := fExternalValue;
	END_IF
	
	4: //pressure difference control
	fAct := localState.fPressureDifference;
	
	5: //proportional pressure control
	fAct := localState.fPressureDifference;
	
	6: //thermal power
	fAct := fThermalPowerExternal;
END_CASE

//switch setpoint and actual value depending on heating or cooling mode
CASE nControlMode OF
	1: //flow is heated
	fSetpointValue := fAct;
	fActualValue := fSetPoint;	

	2: //flow is cooled
	fSetpointValue := fSetPoint;	
	fActualValue := fAct;
	
	3: //temperature difference
	fSetpointValue := ABS(fAct);
	fActualValue := ABS(fSetPoint);
	
	4: //pressure difference control
	fSetpointValue := fSetPoint;
	fActualValue := fAct;
	
	5: //proportional pressure control
	//calculate linear curve depending on fSetPoint
	fSetpointValue := (fSetPoint-(fSetPoint/2))/((fSetPoint-localDefaultParameters.fMaximumPressureDifference+(localDefaultParameters.fMaximumPressureDifference/(localDefaultParameters.fMaximumVolumeFlowRate-localDefaultParameters.fNominalVolumeFlowRate))*localDefaultParameters.fMaximumVolumeFlowRate)*((localDefaultParameters.fNominalVolumeFlowRate-localDefaultParameters.fMaximumVolumeFlowRate)/localDefaultParameters.fMaximumPressureDifference));
	fActualValue := fAct;
	
	6: //thermal power
	fSetpointValue := ABS(fSetPoint);
	fActualValue := ABS(fAct);
END_CASE

PI_Controller (
		fSetpointValue	:= fSetpointValue,
		fActualValue	:= fActualValue,
		fManSyncValue	:= 0,
		bSync			:= FALSE,
		eMode			:= 2, (* mode active *)
		bHold			:= FALSE,
		stParams		:= PI_Controller_Parameters);

//output of PI controller is not used in frequency control mode
CASE nControlMode OF
	0:
	fSetPoint_controlled := fSetPoint;
ELSE	
	fSetPoint_controlled := LREAL_TO_REAL(PI_Controller.fOut);
END_CASE
END_METHOD

METHOD PRIVATE SelectLocalControlMode : BOOL
VAR_INPUT
END_VAR
IF control.bManualModeActivated THEN
	nControlMode := localSetParameters.nControlModeManual;
ELSIF control.bAlgorithmModeActivated AND bAlgorithmPermission THEN
	nControlMode := localSetParameters.nControlModeAlgorithm;
ELSE
	nControlMode := nControlModeAutomatic;
END_IF
END_METHOD

METHOD PROTECTED  SetSetPointLimits : BOOL
VAR_INPUT
END_VAR
CASE nControlMode OF
	0: //constant speed
	aSetPointLimits := localDefaultParameters.aSetPointLimits_constantSpeed;

	1,2,3: //temperature mode
	aSetPointLimits := localDefaultParameters.aSetPointLimits_Temperature;
	
	4,5: //pressure
	aSetPointLimits := localDefaultParameters.aSetPointLimits_Pressure;
END_CASE
END_METHOD

METHOD SetState_Profibus : BOOL
VAR_INPUT
END_VAR
VAR
END_VAR
//setpoint state
setPointState.fSetPoint := fSetPoint;
setPointState.aSetPointLimits := aSetPointLimits;
CASE nControlMode OF
	0: //position mode
	setPointState.sSetPointUnit := 'percent';
	
	1,2: //constant temperature
	setPointState.sSetPointUnit := 'degreeC';
	
	3: //temperature difference
	setPointState.sSetPointUnit := 'K';
END_CASE

//output
controlModule0Bits[0] := TRUE; //Remote control
controlModule0Bits[1] := bSetStatusOn;//bit for switching on pump
controlModule0Bits[2] := localSetParameters.bReset; //bit to reset errors and warnings

ControlModule_OUT[0] := ConvertBitToByte(dataBit:=controlModule0Bits);
ControlModule_OUT[1] := 1;
ControlModule_OUT[2] := 0;
tmp := DWORD_TO_HEXSTR(DINT_TO_DWORD(TRUNC(fSetPoint_controlled*100)),4,TRUE);
ControlModule_OUT[3] := HEXCHRNIBBLE_TO_BYTE(MID(tmp,1,1))*16 + HEXCHRNIBBLE_TO_BYTE(MID(tmp,1,2));
ControlModule_OUT[4] := HEXCHRNIBBLE_TO_BYTE(MID(tmp,1,3))*16 + HEXCHRNIBBLE_TO_BYTE(MID(tmp,1,4));
END_METHOD

PROPERTY ST_DefaultParameters : REFERENCE TO ST_PumpGrundfosMagna3DefaultParameters
SET
localDefaultParameters := ST_DefaultParameters;
END_SET
END_PROPERTY

END_FUNCTION_BLOCK

// ---- POUs/3 Utilities/2 Profibus/BufferUdintToReal.TcPOU
FUNCTION BufferUdintToReal : REAL
VAR_INPUT
	raw_input :UDINT;
END_VAR
VAR
	temp : DWORD;
END_VAR

temp := UDINT_TO_DWORD(raw_input);
BufferUdintToReal := DWORD_TO_REAL(temp);
temp := BE32_TO_HOST(temp);
MEMCPY(ADR(BufferUdintToReal), ADR(temp), SIZEOF(temp));

END_FUNCTION

// ---- POUs/1 Actors/FB_MixingValve.TcPOU
FUNCTION_BLOCK FB_MixingValve EXTENDS FB_ActuatorContinous
VAR_INPUT
	nControlModeAutomatic : E_MixingValveControlMode;
	fTemperatureExternal : REAL; //External temperature in °C
	fThermalPowerExternal : REAL; //external heat power in kW
END_VAR
VAR_OUTPUT
END_VAR
VAR	
	{attribute 'OPC.UA.DA' := '1'}
	localSetParameters 			: ST_MixingValveSetParameters;
	
	//default parameters
	localDefaultParameters 		: ST_MixingValveDefaultParameters;	

	//analog converters for 0 - 10 V i/o signals
	InputConverter 				: FB_AnalogInput(fLowerLimit := 0, fUpperLimit := 100);
	OutputConverter 			: FB_AnalogOutput(fLowerLimit := 0, fUpperLimit := 100);
	
	//I/O Links
	nSetPoint_OUT		AT %Q* : INT; //Set position linked to terminal
	nOperatingPoint_IN 	AT %I* : INT; //Actual valve position linked to terminal
	
	//internal variables
	nControlMode				: E_MixingValveControlMode;	
	fSetPoint_internal 			: REAL; //internal, control mode depending setpoint between 0.0 and 100.0
	
	//controllers
	PI_Controller_Heating		: FB_CTRL_PI; 
	PI_Controller_Cooling		: FB_CTRL_PI;
	PI_Controller_ThermalPower	: FB_CTRL_PI;
	PI_Controller_Parameters 	: ST_CTRL_PI_PARAMS;
END_VAR

MAIN();
SelectLocalControlMode();
LocalControl();
InputConverter(nValue := nOperatingPoint_IN, fOffset := localDefaultParameters.fOffsetTerminal);
OutputConverter(fValue := fSetPoint_internal);

METHOD GetState_AI : BOOL
VAR_INPUT
END_VAR
IF localDefaultParameters.bFeedbackSignal = TRUE THEN //Set operating point if there is a feedback signal 
	setPointState.fOperatingPoint := InputConverter.fValue;
	fOperatingPoint := setPointState.fOperatingPoint;
	setPointState.sOperatingPointUnit := 'percent';
	IF setPointState.fOperatingPoint > 0 THEN //Set control state if valve is open
		controlState.bStatusOn := TRUE;
		bStatusOn := TRUE;
	ELSE
		controlState.bStatusOn := FALSE;
		bStatusOn := FALSE;
	END_IF
END_IF;
END_METHOD

METHOD PRIVATE LocalControl : BOOL
VAR_INPUT
END_VAR
VAR
END_VAR
//set control parameters
PI_Controller_Parameters.fKp 				:= localDefaultParameters.fControllerAmplification;
PI_Controller_Parameters.tTn 				:= localDefaultParameters.tControllerIntegralTime;
PI_Controller_Parameters.fOutMaxLimit		:= localDefaultParameters.fOutMaxLimit;
PI_Controller_Parameters.fOutMinLimit		:= localDefaultParameters.fOutMinLimit;
PI_Controller_Parameters.tTaskCycleTime		:= localDefaultParameters.tTaskCycleTime;
PI_Controller_Parameters.tCtrlCycleTime		:= localDefaultParameters.tCtrlCycleTime;
PI_Controller_Parameters.bARWOnIPartOnly	:= localDefaultParameters.bARWOnIPartOnly;

IF bSetStatusOn THEN
	CASE nControlMode OF
		0: //position mode
		fSetPoint_internal := fSetPoint;
		
		1: //heating mode
		PI_Controller_Heating (
				fSetpointValue	:= fSetPoint,
				fActualValue	:= fTemperatureExternal,
				fManSyncValue	:= 0,
				bSync			:= FALSE,
				eMode			:= 2, (* mode active *)
				bHold			:= FALSE,
				stParams		:= PI_Controller_Parameters);
		fSetPoint_internal := LREAL_TO_REAL(PI_Controller_Heating.fOut);
				
		2: //cooling mode
		PI_Controller_Cooling (
			fSetpointValue	:= fTemperatureExternal,
			fActualValue	:= fSetPoint,
			fManSyncValue	:= 0,
			bSync			:= FALSE,
			eMode			:= 2, (* mode active *)
			bHold			:= FALSE,
			stParams		:= PI_Controller_Parameters);
		fSetPoint_internal := LREAL_TO_REAL(PI_Controller_Cooling.fOut);
		
		3: //thermal power
		PI_Controller_ThermalPower (
			fSetpointValue	:= ABS(fSetPoint),
			fActualValue	:= ABS(fThermalPowerExternal),
			fManSyncValue	:= 0,
			bSync			:= FALSE,
			eMode			:= 2, (* mode active *)
			bHold			:= FALSE,
			stParams		:= PI_Controller_Parameters);
		fSetPoint_internal := LREAL_TO_REAL(PI_Controller_ThermalPower.fOut);
	END_CASE
ELSE
	fSetPoint_internal := localDefaultParameters.fDefaultPosition;
END_IF
END_METHOD

METHOD PRIVATE SelectLocalControlMode : BOOL
VAR_INPUT
END_VAR
IF control.bManualModeActivated THEN
	nControlMode := localSetParameters.nControlModeManual;
ELSIF control.bAlgorithmModeActivated AND bAlgorithmPermission THEN
	nControlMode := localSetParameters.nControlModeAlgorithm;
ELSE
	nControlMode := nControlModeAutomatic;
END_IF
END_METHOD

METHOD PROTECTED  SetSetPointLimits : BOOL
VAR_INPUT
END_VAR
CASE nControlMode OF
	0: //position mode
	aSetPointLimits := localDefaultParameters.aSetPointLimitsPosition;

	1: //heating mode
	aSetPointLimits := localDefaultParameters.aSetPointLimitsTemperature;
	
	2: //cooling mode
	aSetPointLimits := localDefaultParameters.aSetPointLimitsTemperature;
	
	3: //themal power
	aSetPointLimits := localDefaultParameters.aSetPointLimitsThermalPower;
END_CASE
END_METHOD

METHOD SetState_AO : BOOL
VAR
END_VAR
setPointState.fSetPoint := fSetPoint;
setPointState.aSetPointLimits := aSetPointLimits;
CASE nControlMode OF
	0: //position mode
	setPointState.sSetPointUnit := 'percent';
	
	1: //heating mode
	setPointState.sSetPointUnit := 'degreeC';
	
	2: //cooling mode
	setPointState.sSetPointUnit := 'degreeC';
	
	3: //thermal power mode
	setPointState.sSetPointUnit := 'kW';

END_CASE

nSetPoint_OUT := OutputConverter.nValue;  //converts real setpoint for terminal
END_METHOD

PROPERTY ST_DefaultParameters : REFERENCE TO ST_MixingValveDefaultParameters
SET
localDefaultParameters := ST_DefaultParameters;
END_SET
END_PROPERTY

END_FUNCTION_BLOCK

// ---- POUs/3 Utilities/1 AI_AO/FB_AnalogOutput.TcPOU
FUNCTION_BLOCK FB_AnalogOutput
VAR_INPUT
END_VAR
VAR_INPUT
	fValue		: REAL; //input value	
END_VAR
VAR_OUTPUT
	nValue 		: INT; //converted value
END_VAR
VAR
	fUpperLimit : REAL; //upper limit of value range
	fLowerLimit : REAL; //lower limit of value range
END_VAR

// conversion from Bit value to actual value
nValue := REAL_TO_INT((fValue-fLowerLimit)/(fUpperLimit-fLowerLimit)*32767);

METHOD FB_init : BOOL
VAR_INPUT
	bInitRetains : BOOL; // if TRUE, the retain variables are initialized (warm start / cold start)
	bInCopyCode : BOOL;  // if TRUE, the instance afterwards gets moved into the copy code (online change)
	fUpperLimit : REAL; //upper limit of value range
	fLowerLimit : REAL; //lower limit of value range
END_VAR
//copy input values to internal variables
THIS^.fUpperLimit := fUpperLimit;
THIS^.fLowerLimit := fLowerLimit;
END_METHOD

END_FUNCTION_BLOCK

// ---- POUs/2 Sensors/FB_MollineC3HeatCounter.TcPOU
FUNCTION_BLOCK FB_MollineC3HeatCounter
VAR_INPUT
	aHeatCounterTelegramm : ARRAY[1..cMBUS_MaxTelegrams] OF ST_MBus_Data2;
END_VAR
VAR_OUTPUT
	fFeedTemperature : REAL; //°C
	fReturnTemperature : REAL; //°C
	fVolumeFlowRate : REAL; //m3/h
	fHeatFlowRate : REAL; //kW
END_VAR
VAR
	//default parameters
	localDefaultParameters : ST_MollineC3HeatCounterDefaultParameters;	

	{attribute 'OPC.UA.DA' := '1'}
	sensorState : ST_MollineC3HeatCounterState;
END_VAR

//set sensor state
sensorState.fVolume := STRING_TO_REAL(aHeatCounterTelegramm[1].arrData[3].sValue);
sensorState.fFeedTemperature := STRING_TO_REAL(aHeatCounterTelegramm[1].arrData[8].sValue);
sensorState.fReturnTemperature := STRING_TO_REAL(aHeatCounterTelegramm[1].arrData[9].sValue);
sensorState.fVolumeFlowRate := STRING_TO_REAL(aHeatCounterTelegramm[1].arrData[6].sValue);
sensorState.fHeatEnergy := STRING_TO_REAL(aHeatCounterTelegramm[1].arrData[2].sValue)/1000000;
sensorState.fTemperatureDifference := STRING_TO_REAL(aHeatCounterTelegramm[1].arrData[10].sValue);

//calculate fHeatFlowRate because heat meter does not measure negative flows
sensorState.fHeatFlowRate := sensorState.fVolumeFlowRate/3.6*localDefaultParameters.fSpecificHeatCapacity*sensorState.fTemperatureDifference;

//set outputs
fFeedTemperature := sensorState.fFeedTemperature;
fReturnTemperature := sensorState.fReturnTemperature;
fVolumeFlowRate := sensorState.fVolumeFlowRate;
fHeatFlowRate := sensorState.fHeatFlowRate;

PROPERTY ST_DefaultParameters : REFERENCE TO ST_MollineC3HeatCounterDefaultParameters
SET
localDefaultParameters := ST_DefaultParameters;
END_SET
END_PROPERTY

END_FUNCTION_BLOCK

// ---- POUs/2 Sensors/FB_TemperatureSensor.TcPOU
FUNCTION_BLOCK FB_TemperatureSensor EXTENDS FB_Sensor
VAR_INPUT
END_VAR
VAR_OUTPUT
	fTemperature : REAL; //measured temperature in degreeC
END_VAR
VAR	
	//I/O-Links
	temperature_IN AT %I* : INT;
END_VAR

METHOD GetState_AI : BOOL
VAR_INPUT
END_VAR
VAR
END_VAR
// conversion with 0.01 resolution
fTemperature := (INT_TO_REAL(temperature_IN))*0.01;

//sensor state
sensorState.fValue := fTemperature;
sensorState.sUnit := 'degreeC';
END_METHOD

END_FUNCTION_BLOCK

// ---- POUs/3 Utilities/0 Base/Limiter.TcPOU
FUNCTION Limiter : BOOL
VAR_INPUT
	fInput : REAL;
	fUpperLimit : REAL;
	fLowerLimit : REAL;
END_VAR
VAR
END_VAR

IF fInput <= fUpperLimit AND fInput >= fLowerLimit THEN
	Limiter := TRUE;
ELSE
	Limiter := FALSE;		
END_IF

END_FUNCTION
